FUNCTION_BLOCK FB_XMLRead
VAR
	fbXmlSrvRead				:	FB_XmlSrvRead;
	fbXmlSrvReadByName			:	FB_XmlSrvReadByName;
	xExecute					:	BOOL:=FALSE;
	
	sFilePath					:T_MaxString := 'C:\Users\Ignacy\Downloads\PCM_Template.xml';
	sXPath						:T_MaxString := '/ProductionChange/MESSAGEHEADER';
	sXPath1						:T_MaxString := '/ProductionChange/PRODUCTINFORMATION';
	iStep						:INT;
	st_productionchange			:ST_ProductionChange;
END_VAR

fbXmlSrvRead(
   		sNetId := '', 
    	pSymAddr := ADR(st_productionchange.MESSAGEHEADER),
  		cbSymSize := SIZEOF(st_productionchange.MESSAGEHEADER),
    	sFilePath := sFilePath,
    	sXPath := sXPath,
    	bExecute := xExecute);
fbXmlSrvRead(
    	sNetId := '', 
    	pSymAddr := ADR(st_productionchange.PRODUCTINFORMATION),
   		cbSymSize := SIZEOF(st_productionchange.PRODUCTINFORMATION),
    	sFilePath := sFilePath,
    	sXPath := sXPath1,
    	bExecute := xExecute);

	IF NOT xExecute THEN
  	  xExecute := TRUE;
	END_IF;

	IF NOT fbXmlSrvRead.bBusy AND xExecute THEN
   	 xExecute := FALSE; 
	END_IF;

END_FUNCTION_BLOCK

(* stored: Version 1.1.0.1, ProductVersion 3.1.4024.13
   POU FB_XMLRead: Id {cbbbc43d-edf9-4a81-a73e-eb6873779509}, SpecialFunc None *)
